(* Logix 5000 project; controller Generic 1768-L43 rev 16.2; software revision 15.01; part 2 of 10 *)
(* tags used below, declared in another part *)
   EL_CTRL_2 : UDT_AxisHistory_CTRL;
   EL_CTRL_3 : UDT_AxisHistory_CTRL;
   EL_CTRL_4 : UDT_AxisHistory_CTRL;
   EventLog_N2 : UDT_AxisHistory_DLM[51];
   EventLog_N3 : UDT_AxisHistory_DLM[51];
   EventLog_N4 : UDT_AxisHistory_DLM[51];
   LogLength : DINT;
   Motion_Group : ALIAS FOR MotionGroup;
   Servo_Axis_Node_2 : ALIAS FOR AXIS_02;
   Servo_Axis_Node_3 : ALIAS FOR AXIS_03;
   Servo_Axis_Node_4 : ALIAS FOR AXIS_04;
(* AXIS_EventLog, continued *)

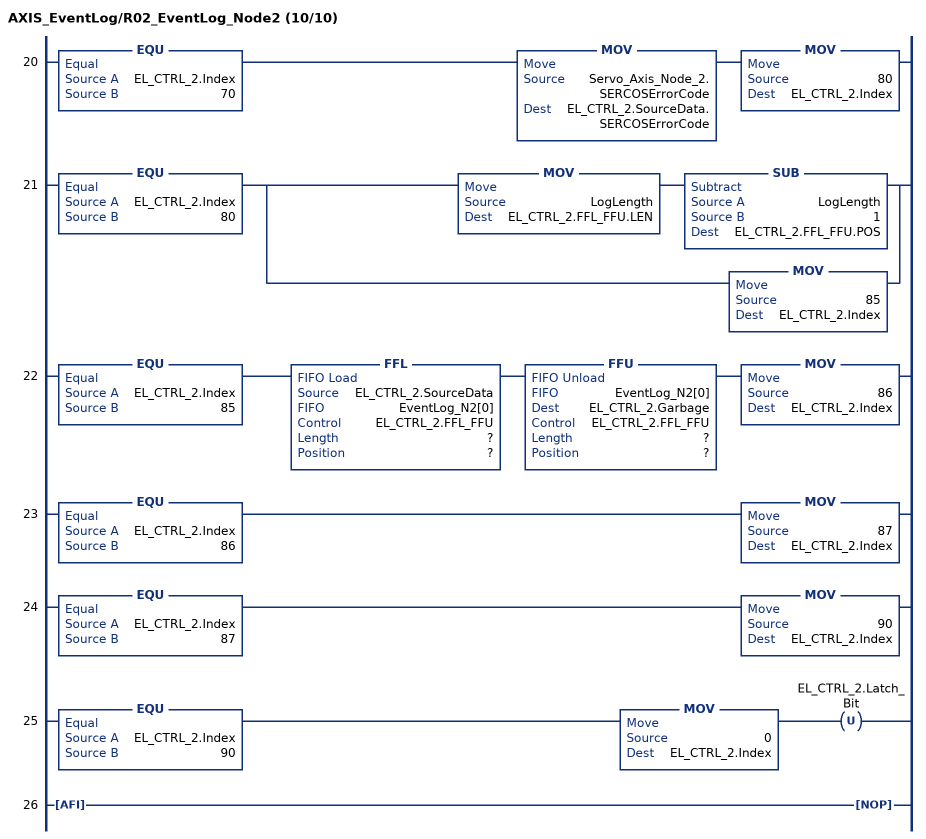
   [picture p36: AXIS_EventLog/R02_EventLog_Node2 rungs 20-26]
   20: EQU(EL_CTRL_2.Index,70)MOV(Servo_Axis_Node_2.SERCOSErrorCode,EL_CTRL_2.SourceData.SERCOSErrorCode)MOV(80,EL_CTRL_2.Index);
   21: EQU(EL_CTRL_2.Index,80)[MOV(LogLength,EL_CTRL_2.FFL_FFU.LEN) SUB(LogLength,1,EL_CTRL_2.FFL_FFU.POS) ,MOV(85,EL_CTRL_2.Index) ];
   22: EQU(EL_CTRL_2.Index,85)FFL(EL_CTRL_2.SourceData,EventLog_N2[0],EL_CTRL_2.FFL_FFU,?,?)FFU(EventLog_N2[0],EL_CTRL_2.Garbage,EL_CTRL_2.FFL_FFU,?,?)MOV(86,EL_CTRL_2.Index);
   23: EQU(EL_CTRL_2.Index,86)MOV(87,EL_CTRL_2.Index);
   24: EQU(EL_CTRL_2.Index,87)MOV(90,EL_CTRL_2.Index);
   25: EQU(EL_CTRL_2.Index,90)MOV(0,EL_CTRL_2.Index)OTU(EL_CTRL_2.Latch_Bit);
   26: AFI()NOP();
END_ROUTINE

ROUTINE R03_EventLog_Node3   (* ladder *)
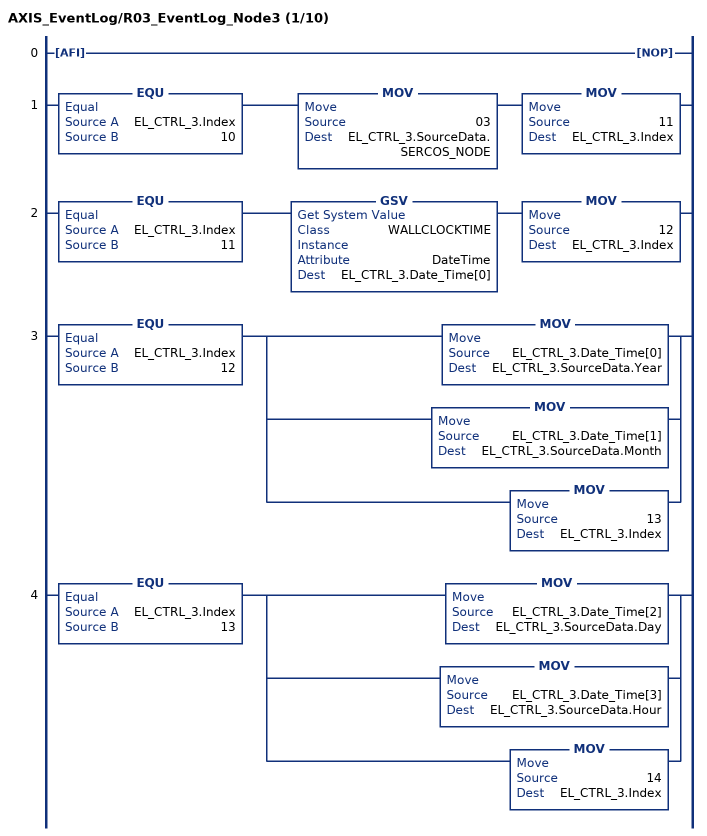
   0: AFI()NOP();
   1: EQU(EL_CTRL_3.Index,10)MOV(03,EL_CTRL_3.SourceData.SERCOS_NODE)MOV(11,EL_CTRL_3.Index);
   2: EQU(EL_CTRL_3.Index,11)GSV(WALLCLOCKTIME,,DateTime,EL_CTRL_3.Date_Time[0])MOV(12,EL_CTRL_3.Index);
   3: EQU(EL_CTRL_3.Index,12)[MOV(EL_CTRL_3.Date_Time[0],EL_CTRL_3.SourceData.Year) ,MOV(EL_CTRL_3.Date_Time[1],EL_CTRL_3.SourceData.Month) ,MOV(13,EL_CTRL_3.Index) ];
   4: EQU(EL_CTRL_3.Index,13)[MOV(EL_CTRL_3.Date_Time[2],EL_CTRL_3.SourceData.Day) ,MOV(EL_CTRL_3.Date_Time[3],EL_CTRL_3.SourceData.Hour) ,MOV(14,EL_CTRL_3.Index) ];
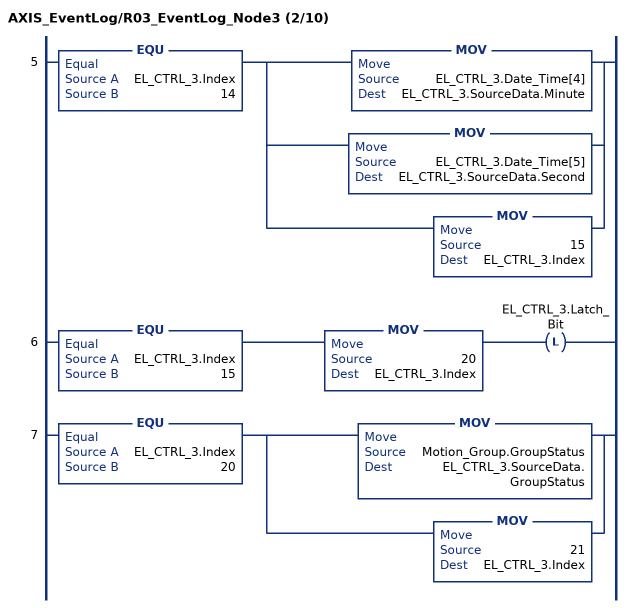
   5: EQU(EL_CTRL_3.Index,14)[MOV(EL_CTRL_3.Date_Time[4],EL_CTRL_3.SourceData.Minute) ,MOV(EL_CTRL_3.Date_Time[5],EL_CTRL_3.SourceData.Second) ,MOV(15,EL_CTRL_3.Index) ];
   6: EQU(EL_CTRL_3.Index,15)MOV(20,EL_CTRL_3.Index)OTL(EL_CTRL_3.Latch_Bit);
   7: EQU(EL_CTRL_3.Index,20)[MOV(Motion_Group.GroupStatus,EL_CTRL_3.SourceData.GroupStatus) ,MOV(21,EL_CTRL_3.Index) ];
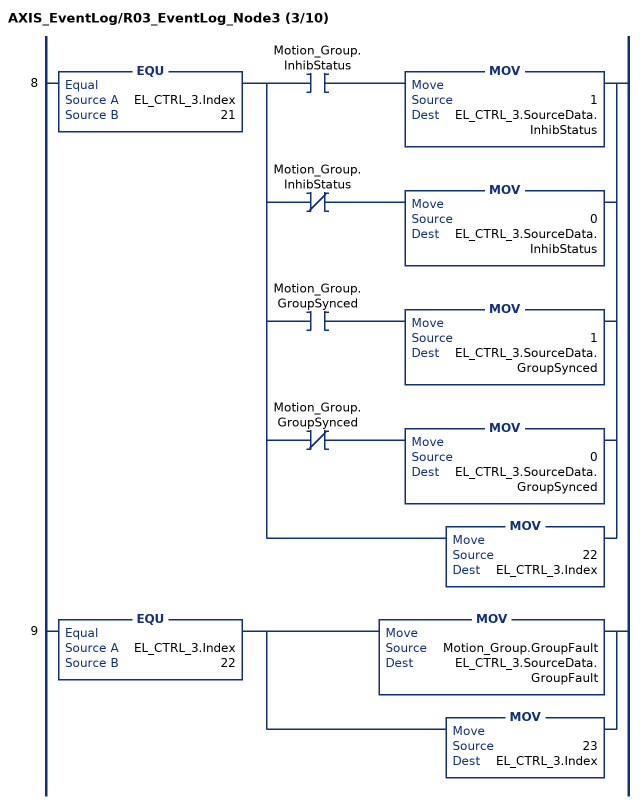
   8: EQU(EL_CTRL_3.Index,21)[XIC(Motion_Group.InhibStatus) MOV(1,EL_CTRL_3.SourceData.InhibStatus) ,XIO(Motion_Group.InhibStatus) MOV(0,EL_CTRL_3.SourceData.InhibStatus) ,XIC(Motion_Group.GroupSynced) MOV(1,EL_CTRL_3.SourceData.GroupSynced) ,XIO(Motion_Group.GroupSynced) MOV(0,EL_CTRL_3.SourceData.GroupSynced) ,MOV(22,EL_CTRL_3.Index) ];
   9: EQU(EL_CTRL_3.Index,22)[MOV(Motion_Group.GroupFault,EL_CTRL_3.SourceData.GroupFault) ,MOV(23,EL_CTRL_3.Index) ];
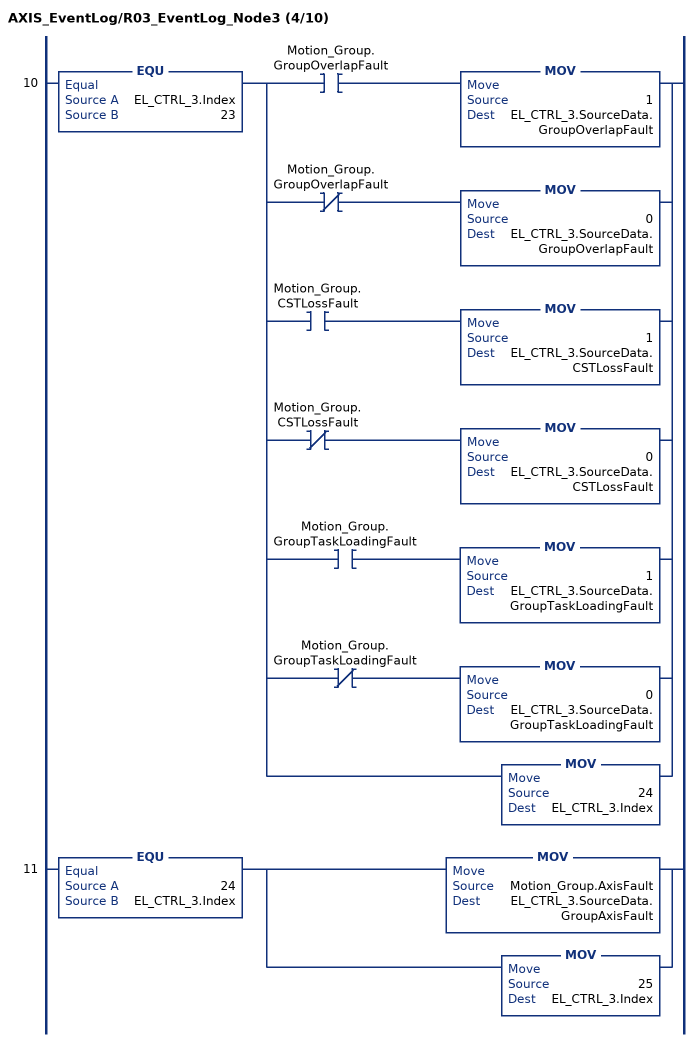
   10: EQU(EL_CTRL_3.Index,23)[XIC(Motion_Group.GroupOverlapFault) MOV(1,EL_CTRL_3.SourceData.GroupOverlapFault) ,XIO(Motion_Group.GroupOverlapFault) MOV(0,EL_CTRL_3.SourceData.GroupOverlapFault) ,XIC(Motion_Group.CSTLossFault) MOV(1,EL_CTRL_3.SourceData.CSTLossFault) ,XIO(Motion_Group.CSTLossFault) MOV(0,EL_CTRL_3.SourceData.CSTLossFault) ,XIC(Motion_Group.GroupTaskLoadingFault) MOV(1,EL_CTRL_3.SourceData.GroupTaskLoadingFault) ,XIO(Motion_Group.GroupTaskLoadingFault) MOV(0,EL_CTRL_3.SourceData.GroupTaskLoadingFault) ,MOV(24,EL_CTRL_3.Index) ];
   11: EQU(24,EL_CTRL_3.Index)[MOV(Motion_Group.AxisFault,EL_CTRL_3.SourceData.GroupAxisFault) ,MOV(25,EL_CTRL_3.Index) ];
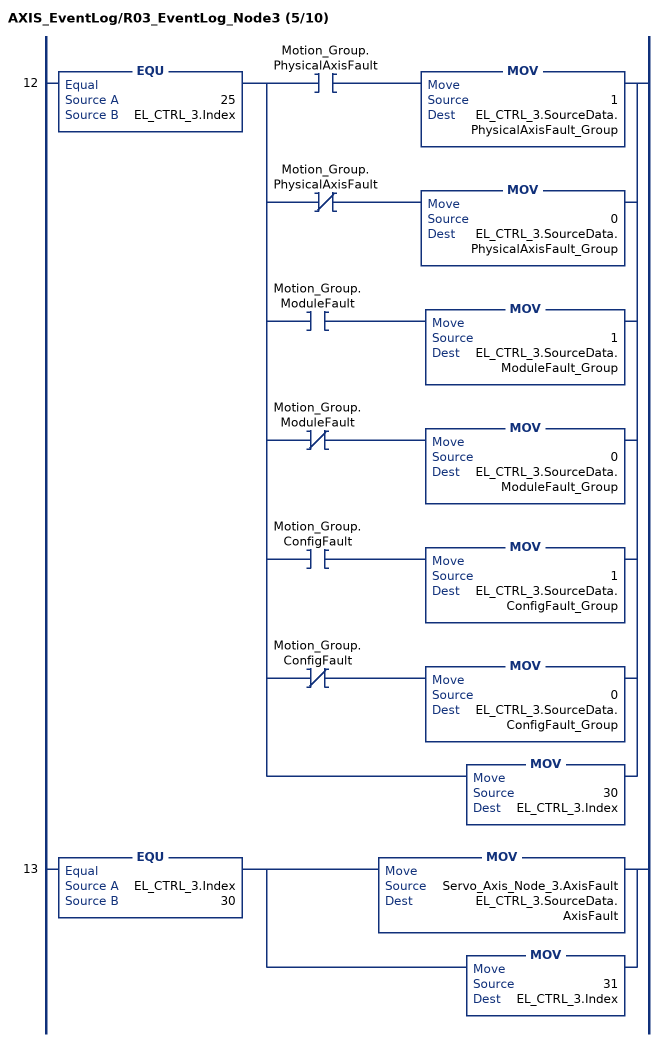
   12: EQU(25,EL_CTRL_3.Index)[XIC(Motion_Group.PhysicalAxisFault) MOV(1,EL_CTRL_3.SourceData.PhysicalAxisFault_Group) ,XIO(Motion_Group.PhysicalAxisFault) MOV(0,EL_CTRL_3.SourceData.PhysicalAxisFault_Group) ,XIC(Motion_Group.ModuleFault) MOV(1,EL_CTRL_3.SourceData.ModuleFault_Group) ,XIO(Motion_Group.ModuleFault) MOV(0,EL_CTRL_3.SourceData.ModuleFault_Group) ,XIC(Motion_Group.ConfigFault) MOV(1,EL_CTRL_3.SourceData.ConfigFault_Group) ,XIO(Motion_Group.ConfigFault) MOV(0,EL_CTRL_3.SourceData.ConfigFault_Group) ,MOV(30,EL_CTRL_3.Index) ];
   13: EQU(EL_CTRL_3.Index,30)[MOV(Servo_Axis_Node_3.AxisFault,EL_CTRL_3.SourceData.AxisFault) ,MOV(31,EL_CTRL_3.Index) ];
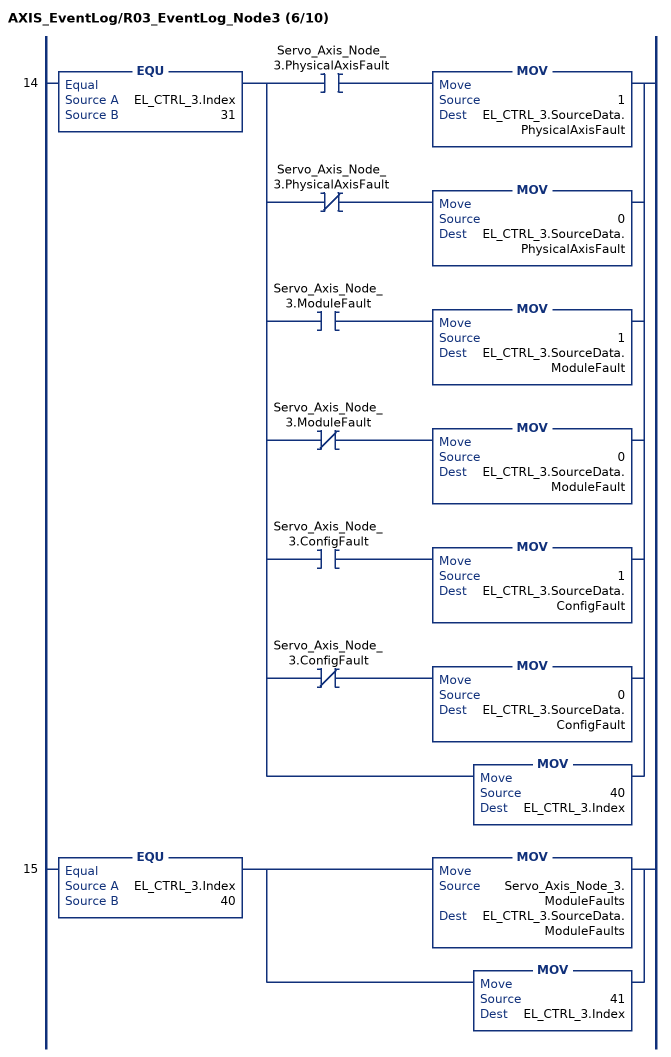
   14: EQU(EL_CTRL_3.Index,31)[XIC(Servo_Axis_Node_3.PhysicalAxisFault) MOV(1,EL_CTRL_3.SourceData.PhysicalAxisFault) ,XIO(Servo_Axis_Node_3.PhysicalAxisFault) MOV(0,EL_CTRL_3.SourceData.PhysicalAxisFault) ,XIC(Servo_Axis_Node_3.ModuleFault) MOV(1,EL_CTRL_3.SourceData.ModuleFault) ,XIO(Servo_Axis_Node_3.ModuleFault) MOV(0,EL_CTRL_3.SourceData.ModuleFault) ,XIC(Servo_Axis_Node_3.ConfigFault) MOV(1,EL_CTRL_3.SourceData.ConfigFault) ,XIO(Servo_Axis_Node_3.ConfigFault) MOV(0,EL_CTRL_3.SourceData.ConfigFault) ,MOV(40,EL_CTRL_3.Index) ];
   15: EQU(EL_CTRL_3.Index,40)[MOV(Servo_Axis_Node_3.ModuleFaults,EL_CTRL_3.SourceData.ModuleFaults) ,MOV(41,EL_CTRL_3.Index) ];
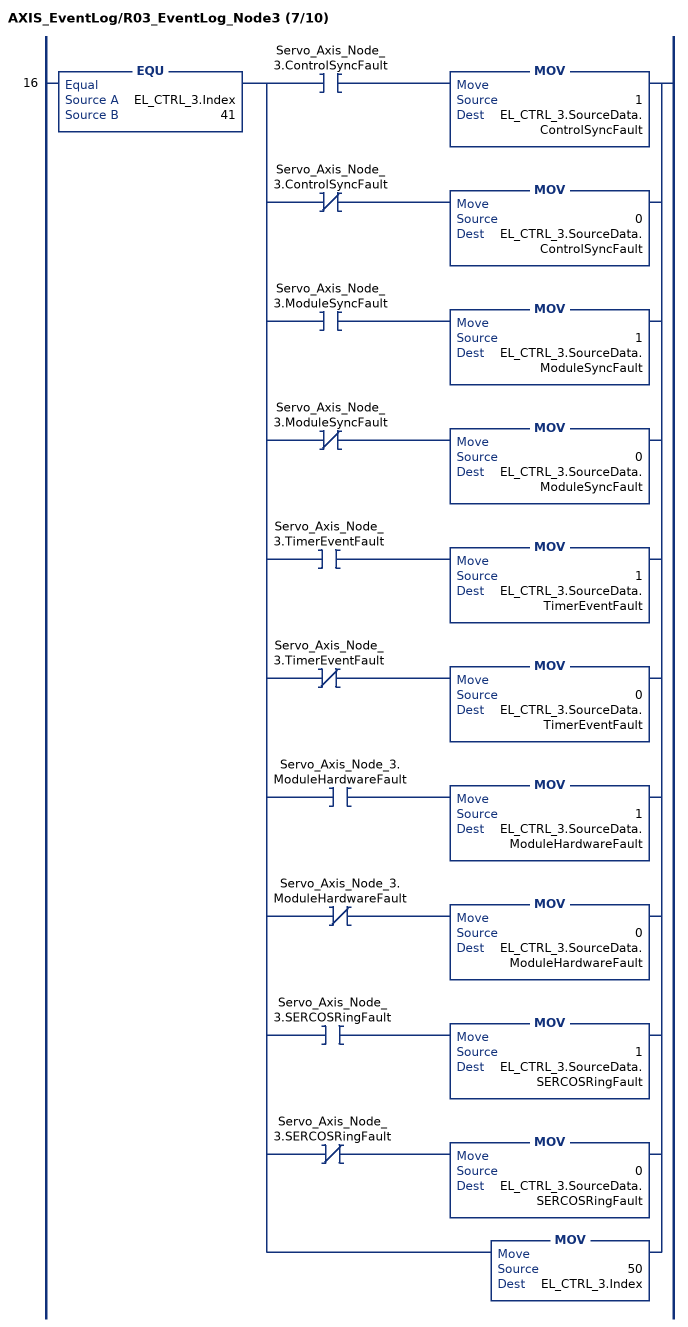
   16: EQU(EL_CTRL_3.Index,41)[XIC(Servo_Axis_Node_3.ControlSyncFault) MOV(1,EL_CTRL_3.SourceData.ControlSyncFault) ,XIO(Servo_Axis_Node_3.ControlSyncFault) MOV(0,EL_CTRL_3.SourceData.ControlSyncFault) ,XIC(Servo_Axis_Node_3.ModuleSyncFault) MOV(1,EL_CTRL_3.SourceData.ModuleSyncFault) ,XIO(Servo_Axis_Node_3.ModuleSyncFault) MOV(0,EL_CTRL_3.SourceData.ModuleSyncFault) ,XIC(Servo_Axis_Node_3.TimerEventFault) MOV(1,EL_CTRL_3.SourceData.TimerEventFault) ,XIO(Servo_Axis_Node_3.TimerEventFault) MOV(0,EL_CTRL_3.SourceData.TimerEventFault) ,XIC(Servo_Axis_Node_3.ModuleHardwareFault) MOV(1,EL_CTRL_3.SourceData.ModuleHardwareFault) ,XIO(Servo_Axis_Node_3.ModuleHardwareFault) MOV(0,EL_CTRL_3.SourceData.ModuleHardwareFault) ,XIC(Servo_Axis_Node_3.SERCOSRingFault) MOV(1,EL_CTRL_3.SourceData.SERCOSRingFault) ,XIO(Servo_Axis_Node_3.SERCOSRingFault) MOV(0,EL_CTRL_3.SourceData.SERCOSRingFault) ,MOV(50,EL_CTRL_3.Index) ];
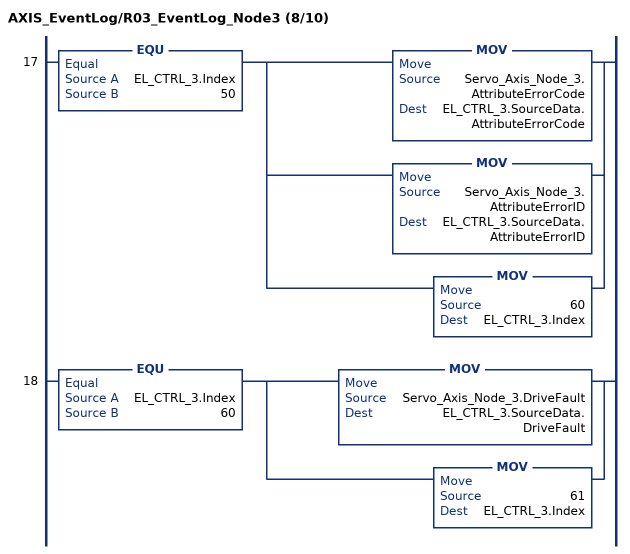
   17: EQU(EL_CTRL_3.Index,50)[MOV(Servo_Axis_Node_3.AttributeErrorCode,EL_CTRL_3.SourceData.AttributeErrorCode) ,MOV(Servo_Axis_Node_3.AttributeErrorID,EL_CTRL_3.SourceData.AttributeErrorID) ,MOV(60,EL_CTRL_3.Index) ];
   18: EQU(EL_CTRL_3.Index,60)[MOV(Servo_Axis_Node_3.DriveFault,EL_CTRL_3.SourceData.DriveFault) ,MOV(61,EL_CTRL_3.Index) ];
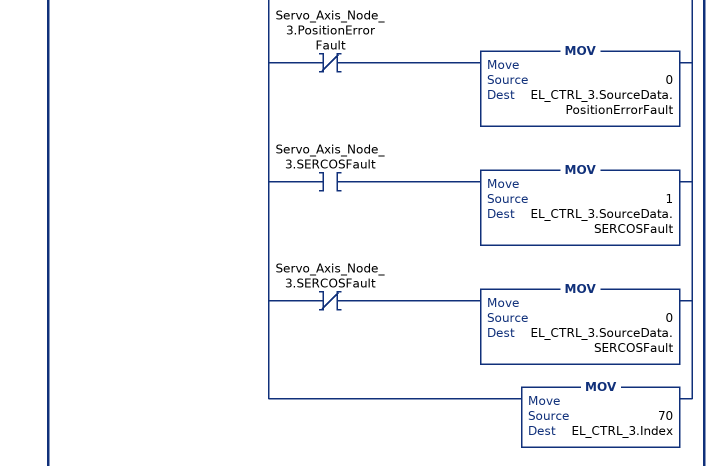
   19: EQU(EL_CTRL_3.Index,61)[XIC(Servo_Axis_Node_3.PosSoftOvertravelFault) MOV(1,EL_CTRL_3.SourceData.PosSoftOvertravelFault) ,XIO(Servo_Axis_Node_3.PosSoftOvertravelFault) MOV(0,EL_CTRL_3.SourceData.PosSoftOvertravelFault) ,XIC(Servo_Axis_Node_3.NegSoftOvertravelFault) MOV(1,EL_CTRL_3.SourceData.NegSoftOvertravelFault) ,XIO(Servo_Axis_Node_3.NegSoftOvertravelFault) MOV(0,EL_CTRL_3.SourceData.NegSoftOvertravelFault) ,XIC(Servo_Axis_Node_3.PosHardOvertravelFault) MOV(1,EL_CTRL_3.SourceData.PosHardOvertravelFault) ,XIO(Servo_Axis_Node_3.PosHardOvertravelFault) MOV(0,EL_CTRL_3.SourceData.PosHardOvertravelFault) ,XIC(Servo_Axis_Node_3.NegHardOvertravelFault) MOV(1,EL_CTRL_3.SourceData.NegHardOvertravelFault) ,XIO(Servo_Axis_Node_3.NegHardOvertravelFault) MOV(0,EL_CTRL_3.SourceData.NegHardOvertravelFault) ,XIC(Servo_Axis_Node_3.MotFeedbackFault) MOV(1,EL_CTRL_3.SourceData.MotFeedbackFault) ,XIO(Servo_Axis_Node_3.MotFeedbackFault) MOV(0,EL_CTRL_3.SourceData.MotFeedbackFault) ,XIC(Servo_Axis_Node_3.MotFeedbackNoiseFault) MOV(1,EL_CTRL_3.SourceData.MotFeedbackNoiseFault) ,XIO(Servo_Axis_Node_3.MotFeedbackNoiseFault) MOV(0,EL_CTRL_3.SourceData.MotFeedbackNoiseFault) ,XIC(Servo_Axis_Node_3.AuxFeedbackFault) MOV(1,EL_CTRL_3.SourceData.AuxFeedbackFault) ,XIO(Servo_Axis_Node_3.AuxFeedbackFault) MOV(0,EL_CTRL_3.SourceData.AuxFeedbackFault) ,XIC(Servo_Axis_Node_3.AuxFeedbackNoiseFault) MOV(1,EL_CTRL_3.SourceData.AuxFeedbackNoiseFault) ,XIO(Servo_Axis_Node_3.AuxFeedbackNoiseFault) MOV(0,EL_CTRL_3.SourceData.AuxFeedbackNoiseFault) ,XIC(Servo_Axis_Node_3.DriveEnableInputFault) MOV(1,EL_CTRL_3.SourceData.DriveEnableInputFault) ,XIO(Servo_Axis_Node_3.DriveEnableInputFault) MOV(0,EL_CTRL_3.SourceData.DriveEnableInputFault) ,XIC(Servo_Axis_Node_3.CommonBusFault) MOV(1,EL_CTRL_3.SourceData.CommonBusFault) ,XIO(Servo_Axis_Node_3.CommonBusFault) MOV(0,EL_CTRL_3.SourceData.CommonBusFault) ,XIC(Servo_Axis_Node_3.PreChargeOverloadFault) MOV(1,EL_CTRL_3.SourceData.PreChargeOverloadFault) ,XIO(Servo_Axis_Node_3.PreChargeOverloadFault) MOV(0,EL_CTRL_3.SourceData.PreChargeOverloadFault) ,XIC(Servo_Axis_Node_3.GroundShortFault) MOV(1,EL_CTRL_3.SourceData.GroundShortFault) ,XIO(Servo_Axis_Node_3.GroundShortFault) MOV(0,EL_CTRL_3.SourceData.GroundShortFault) ,XIC(Servo_Axis_Node_3.DriveHardFault) MOV(1,EL_CTRL_3.SourceData.DriveHardFault) ,XIO(Servo_Axis_Node_3.DriveHardFault) MOV(0,EL_CTRL_3.SourceData.DriveHardFault) ,XIC(Servo_Axis_Node_3.OverSpeedFault) MOV(1,EL_CTRL_3.SourceData.OverSpeedFault) ,XIO(Servo_Axis_Node_3.OverSpeedFault) MOV(0,EL_CTRL_3.SourceData.OverSpeedFault) ,XIC(Servo_Axis_Node_3.OverloadFault) MOV(1,EL_CTRL_3.SourceData.OverloadFault) ,XIO(Servo_Axis_Node_3.OverloadFault) MOV(0,EL_CTRL_3.SourceData.OverloadFault) ,XIC(Servo_Axis_Node_3.DriveOvertempFault) MOV(1,EL_CTRL_3.SourceData.DriveOvertempFault) ,XIO(Servo_Axis_Node_3.DriveOvertempFault) MOV(0,EL_CTRL_3.SourceData.DriveOvertempFault) ,XIC(Servo_Axis_Node_3.MotorOvertempFault) MOV(1,EL_CTRL_3.SourceData.MotorOvertempFault) ,XIO(Servo_Axis_Node_3.MotorOvertempFault) MOV(0,EL_CTRL_3.SourceData.MotorOvertempFault) ,XIC(Servo_Axis_Node_3.DriveCoolingFault) MOV(1,EL_CTRL_3.SourceData.DriveCoolingFault) ,XIO(Servo_Axis_Node_3.DriveCoolingFault) MOV(0,EL_CTRL_3.SourceData.DriveCoolingFault) ,XIC(Servo_Axis_Node_3.DriveControlVoltageFault) MOV(1,EL_CTRL_3.SourceData.DriveControlVoltageFault) ,XIO(Servo_Axis_Node_3.DriveControlVoltageFault) MOV(0,EL_CTRL_3.SourceData.DriveControlVoltageFault) ,XIC(Servo_Axis_Node_3.FeedbackFault) MOV(1,EL_CTRL_3.SourceData.FeedbackFault) ,XIO(Servo_Axis_Node_3.FeedbackFault) MOV(0,EL_CTRL_3.SourceData.FeedbackFault) ,XIC(Servo_Axis_Node_3.CommutationFault) MOV(1,EL_CTRL_3.SourceData.CommutationFault) ,XIO(Servo_Axis_Node_3.CommutationFault) MOV(0,EL_CTRL_3.SourceData.CommutationFault) ,XIC(Servo_Axis_Node_3.DriveOvercurrentFault) MOV(1,EL_CTRL_3.SourceData.DriveOvercurrentFault) ,XIO(Servo_Axis_Node_3.DriveOvercurrentFault) MOV(0,EL_CTRL_3.SourceData.DriveOvercurrentFault) ,XIC(Servo_Axis_Node_3.DriveOvervoltageFault) MOV(1,EL_CTRL_3.SourceData.DriveOvervoltageFault) ,XIO(Servo_Axis_Node_3.DriveOvervoltageFault) MOV(0,EL_CTRL_3.SourceData.DriveOvervoltageFault) ,XIC(Servo_Axis_Node_3.DriveUndervoltageFault) MOV(1,EL_CTRL_3.SourceData.DriveUndervoltageFault) ,XIO(Servo_Axis_Node_3.DriveUndervoltageFault) MOV(0,EL_CTRL_3.SourceData.DriveUndervoltageFault) ,XIC(Servo_Axis_Node_3.PowerPhaseLossFault) MOV(1,EL_CTRL_3.SourceData.PowerPhaseLossFault) ,XIO(Servo_Axis_Node_3.PowerPhaseLossFault) MOV(0,EL_CTRL_3.SourceData.PowerPhaseLossFault) ,XIC(Servo_Axis_Node_3.PositionErrorFault) MOV(1,EL_CTRL_3.SourceData.PositionErrorFault) ,XIO(Servo_Axis_Node_3.PositionErrorFault) MOV(0,EL_CTRL_3.SourceData.PositionErrorFault) ,XIC(Servo_Axis_Node_3.SERCOSFault) MOV(1,EL_CTRL_3.SourceData.SERCOSFault) ,XIO(Servo_Axis_Node_3.SERCOSFault) MOV(0,EL_CTRL_3.SourceData.SERCOSFault) ,MOV(70,EL_CTRL_3.Index) ];
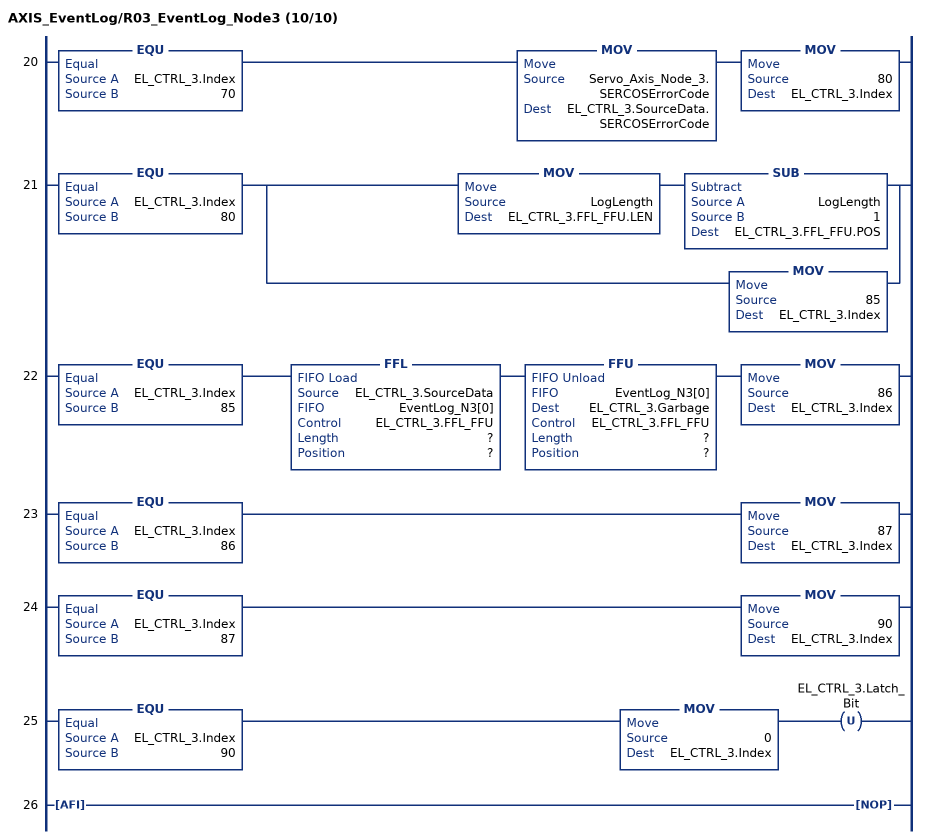
   20: EQU(EL_CTRL_3.Index,70)MOV(Servo_Axis_Node_3.SERCOSErrorCode,EL_CTRL_3.SourceData.SERCOSErrorCode)MOV(80,EL_CTRL_3.Index);
   21: EQU(EL_CTRL_3.Index,80)[MOV(LogLength,EL_CTRL_3.FFL_FFU.LEN) SUB(LogLength,1,EL_CTRL_3.FFL_FFU.POS) ,MOV(85,EL_CTRL_3.Index) ];
   22: EQU(EL_CTRL_3.Index,85)FFL(EL_CTRL_3.SourceData,EventLog_N3[0],EL_CTRL_3.FFL_FFU,?,?)FFU(EventLog_N3[0],EL_CTRL_3.Garbage,EL_CTRL_3.FFL_FFU,?,?)MOV(86,EL_CTRL_3.Index);
   23: EQU(EL_CTRL_3.Index,86)MOV(87,EL_CTRL_3.Index);
   24: EQU(EL_CTRL_3.Index,87)MOV(90,EL_CTRL_3.Index);
   25: EQU(EL_CTRL_3.Index,90)MOV(0,EL_CTRL_3.Index)OTU(EL_CTRL_3.Latch_Bit);
   26: AFI()NOP();
END_ROUTINE

ROUTINE R04_EventLog_Node4   (* ladder *)
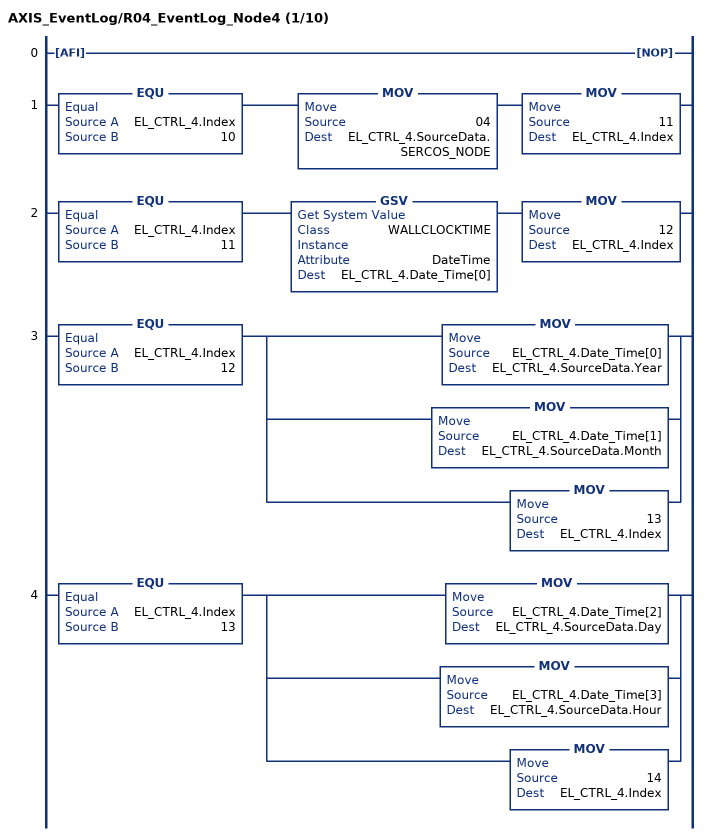
   0: AFI()NOP();
   1: EQU(EL_CTRL_4.Index,10)MOV(04,EL_CTRL_4.SourceData.SERCOS_NODE)MOV(11,EL_CTRL_4.Index);
   2: EQU(EL_CTRL_4.Index,11)GSV(WALLCLOCKTIME,,DateTime,EL_CTRL_4.Date_Time[0])MOV(12,EL_CTRL_4.Index);
   3: EQU(EL_CTRL_4.Index,12)[MOV(EL_CTRL_4.Date_Time[0],EL_CTRL_4.SourceData.Year) ,MOV(EL_CTRL_4.Date_Time[1],EL_CTRL_4.SourceData.Month) ,MOV(13,EL_CTRL_4.Index) ];
   4: EQU(EL_CTRL_4.Index,13)[MOV(EL_CTRL_4.Date_Time[2],EL_CTRL_4.SourceData.Day) ,MOV(EL_CTRL_4.Date_Time[3],EL_CTRL_4.SourceData.Hour) ,MOV(14,EL_CTRL_4.Index) ];
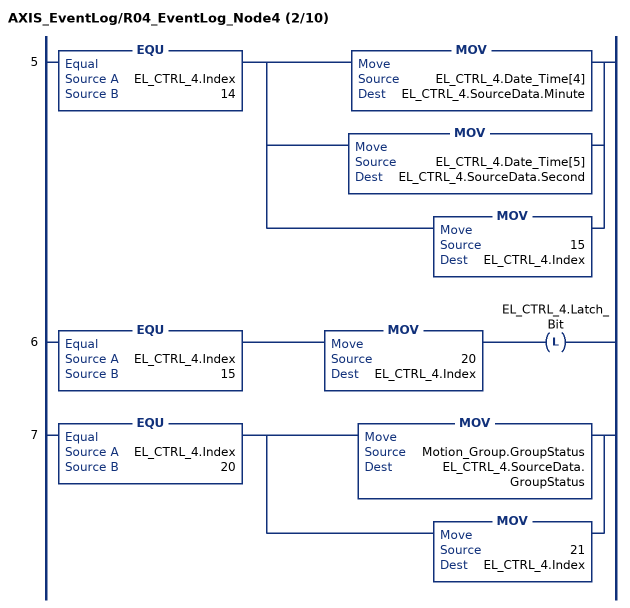
   5: EQU(EL_CTRL_4.Index,14)[MOV(EL_CTRL_4.Date_Time[4],EL_CTRL_4.SourceData.Minute) ,MOV(EL_CTRL_4.Date_Time[5],EL_CTRL_4.SourceData.Second) ,MOV(15,EL_CTRL_4.Index) ];
   6: EQU(EL_CTRL_4.Index,15)MOV(20,EL_CTRL_4.Index)OTL(EL_CTRL_4.Latch_Bit);
   7: EQU(EL_CTRL_4.Index,20)[MOV(Motion_Group.GroupStatus,EL_CTRL_4.SourceData.GroupStatus) ,MOV(21,EL_CTRL_4.Index) ];
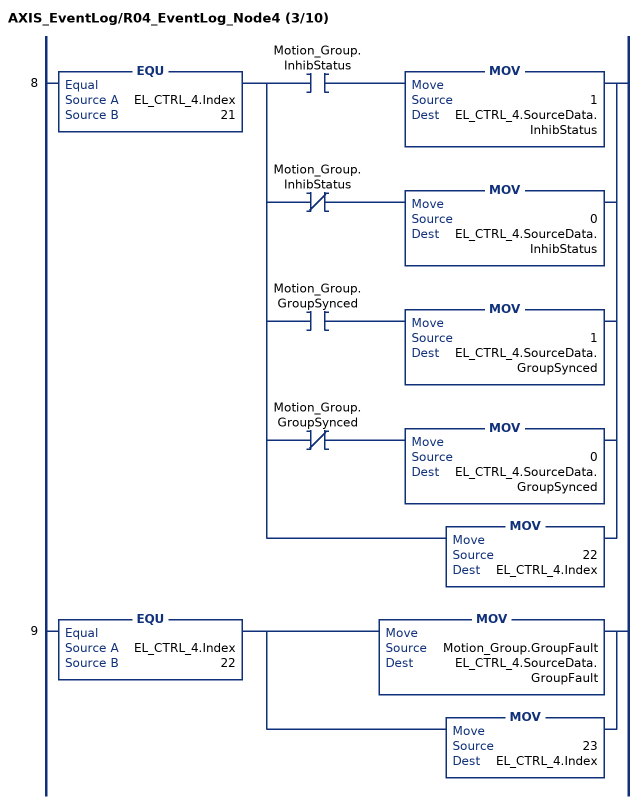
   8: EQU(EL_CTRL_4.Index,21)[XIC(Motion_Group.InhibStatus) MOV(1,EL_CTRL_4.SourceData.InhibStatus) ,XIO(Motion_Group.InhibStatus) MOV(0,EL_CTRL_4.SourceData.InhibStatus) ,XIC(Motion_Group.GroupSynced) MOV(1,EL_CTRL_4.SourceData.GroupSynced) ,XIO(Motion_Group.GroupSynced) MOV(0,EL_CTRL_4.SourceData.GroupSynced) ,MOV(22,EL_CTRL_4.Index) ];
   9: EQU(EL_CTRL_4.Index,22)[MOV(Motion_Group.GroupFault,EL_CTRL_4.SourceData.GroupFault) ,MOV(23,EL_CTRL_4.Index) ];
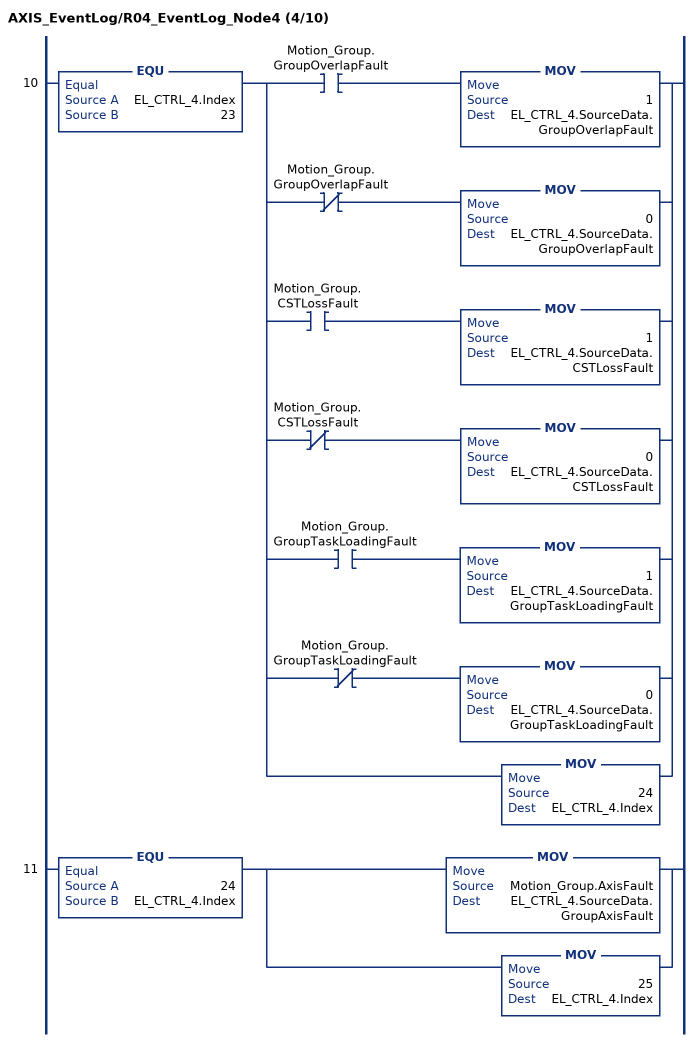
   10: EQU(EL_CTRL_4.Index,23)[XIC(Motion_Group.GroupOverlapFault) MOV(1,EL_CTRL_4.SourceData.GroupOverlapFault) ,XIO(Motion_Group.GroupOverlapFault) MOV(0,EL_CTRL_4.SourceData.GroupOverlapFault) ,XIC(Motion_Group.CSTLossFault) MOV(1,EL_CTRL_4.SourceData.CSTLossFault) ,XIO(Motion_Group.CSTLossFault) MOV(0,EL_CTRL_4.SourceData.CSTLossFault) ,XIC(Motion_Group.GroupTaskLoadingFault) MOV(1,EL_CTRL_4.SourceData.GroupTaskLoadingFault) ,XIO(Motion_Group.GroupTaskLoadingFault) MOV(0,EL_CTRL_4.SourceData.GroupTaskLoadingFault) ,MOV(24,EL_CTRL_4.Index) ];
   11: EQU(24,EL_CTRL_4.Index)[MOV(Motion_Group.AxisFault,EL_CTRL_4.SourceData.GroupAxisFault) ,MOV(25,EL_CTRL_4.Index) ];
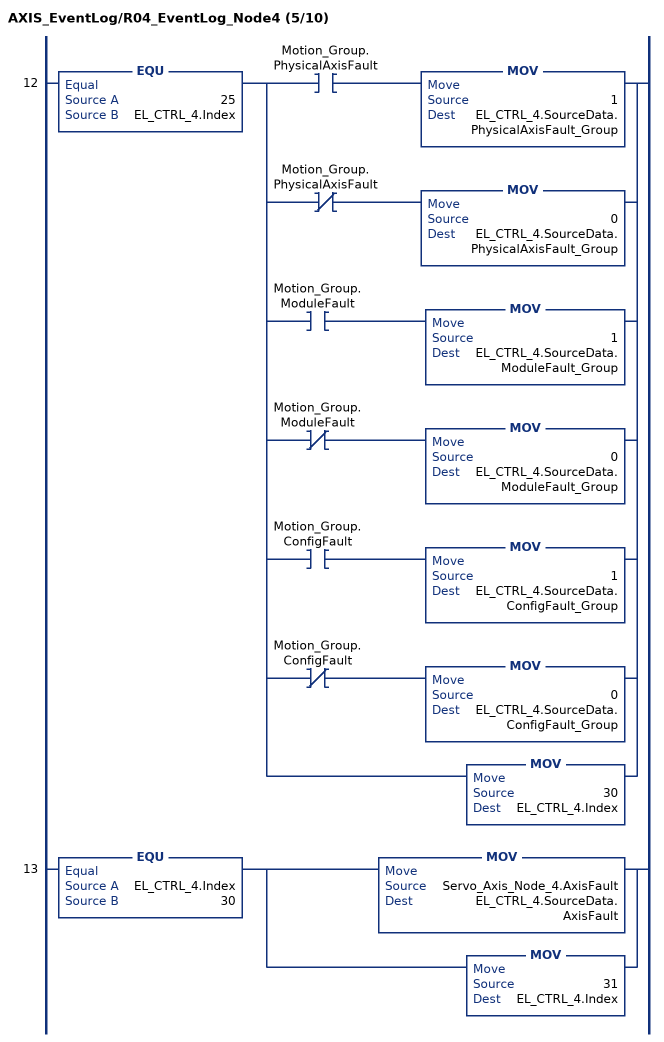
   12: EQU(25,EL_CTRL_4.Index)[XIC(Motion_Group.PhysicalAxisFault) MOV(1,EL_CTRL_4.SourceData.PhysicalAxisFault_Group) ,XIO(Motion_Group.PhysicalAxisFault) MOV(0,EL_CTRL_4.SourceData.PhysicalAxisFault_Group) ,XIC(Motion_Group.ModuleFault) MOV(1,EL_CTRL_4.SourceData.ModuleFault_Group) ,XIO(Motion_Group.ModuleFault) MOV(0,EL_CTRL_4.SourceData.ModuleFault_Group) ,XIC(Motion_Group.ConfigFault) MOV(1,EL_CTRL_4.SourceData.ConfigFault_Group) ,XIO(Motion_Group.ConfigFault) MOV(0,EL_CTRL_4.SourceData.ConfigFault_Group) ,MOV(30,EL_CTRL_4.Index) ];
   13: EQU(EL_CTRL_4.Index,30)[MOV(Servo_Axis_Node_4.AxisFault,EL_CTRL_4.SourceData.AxisFault) ,MOV(31,EL_CTRL_4.Index) ];
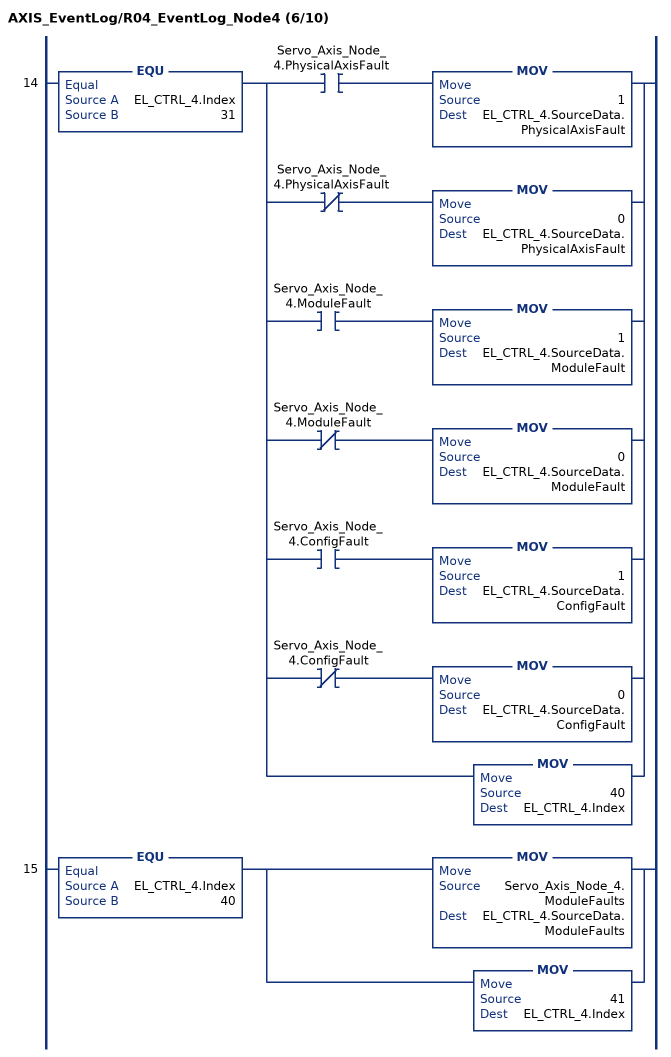
   14: EQU(EL_CTRL_4.Index,31)[XIC(Servo_Axis_Node_4.PhysicalAxisFault) MOV(1,EL_CTRL_4.SourceData.PhysicalAxisFault) ,XIO(Servo_Axis_Node_4.PhysicalAxisFault) MOV(0,EL_CTRL_4.SourceData.PhysicalAxisFault) ,XIC(Servo_Axis_Node_4.ModuleFault) MOV(1,EL_CTRL_4.SourceData.ModuleFault) ,XIO(Servo_Axis_Node_4.ModuleFault) MOV(0,EL_CTRL_4.SourceData.ModuleFault) ,XIC(Servo_Axis_Node_4.ConfigFault) MOV(1,EL_CTRL_4.SourceData.ConfigFault) ,XIO(Servo_Axis_Node_4.ConfigFault) MOV(0,EL_CTRL_4.SourceData.ConfigFault) ,MOV(40,EL_CTRL_4.Index) ];
   15: EQU(EL_CTRL_4.Index,40)[MOV(Servo_Axis_Node_4.ModuleFaults,EL_CTRL_4.SourceData.ModuleFaults) ,MOV(41,EL_CTRL_4.Index) ];
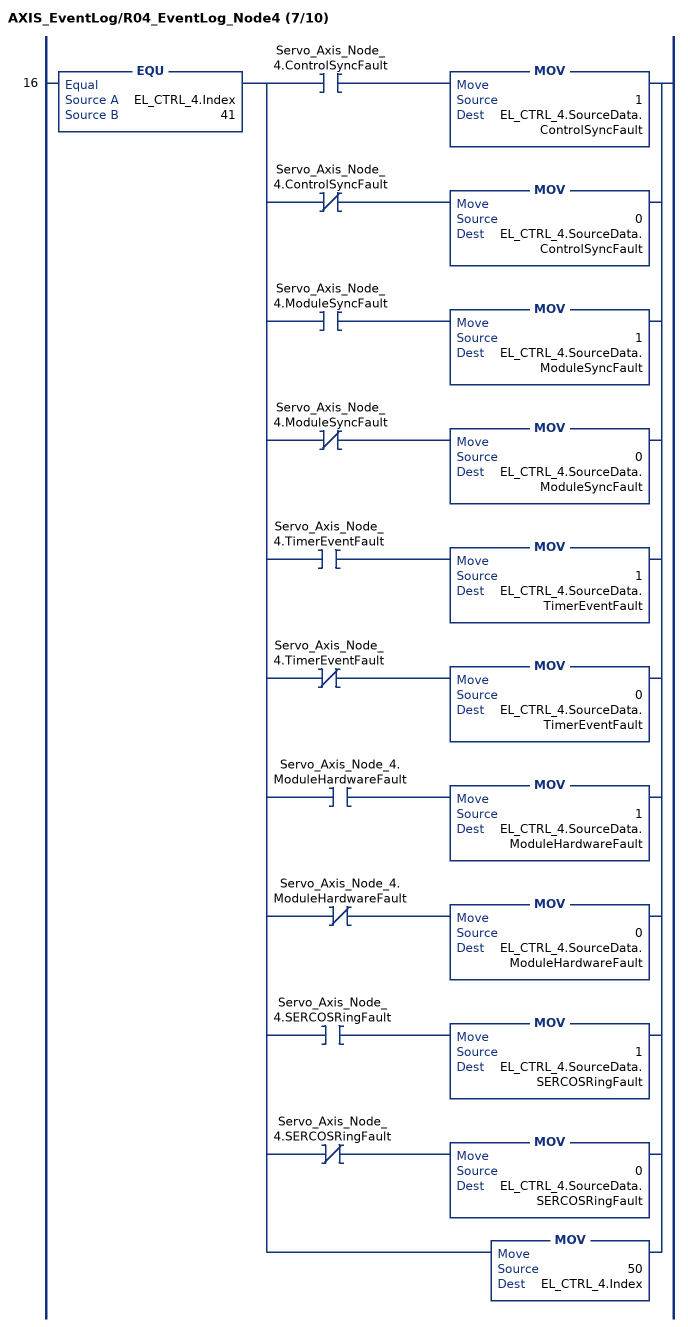
   16: EQU(EL_CTRL_4.Index,41)[XIC(Servo_Axis_Node_4.ControlSyncFault) MOV(1,EL_CTRL_4.SourceData.ControlSyncFault) ,XIO(Servo_Axis_Node_4.ControlSyncFault) MOV(0,EL_CTRL_4.SourceData.ControlSyncFault) ,XIC(Servo_Axis_Node_4.ModuleSyncFault) MOV(1,EL_CTRL_4.SourceData.ModuleSyncFault) ,XIO(Servo_Axis_Node_4.ModuleSyncFault) MOV(0,EL_CTRL_4.SourceData.ModuleSyncFault) ,XIC(Servo_Axis_Node_4.TimerEventFault) MOV(1,EL_CTRL_4.SourceData.TimerEventFault) ,XIO(Servo_Axis_Node_4.TimerEventFault) MOV(0,EL_CTRL_4.SourceData.TimerEventFault) ,XIC(Servo_Axis_Node_4.ModuleHardwareFault) MOV(1,EL_CTRL_4.SourceData.ModuleHardwareFault) ,XIO(Servo_Axis_Node_4.ModuleHardwareFault) MOV(0,EL_CTRL_4.SourceData.ModuleHardwareFault) ,XIC(Servo_Axis_Node_4.SERCOSRingFault) MOV(1,EL_CTRL_4.SourceData.SERCOSRingFault) ,XIO(Servo_Axis_Node_4.SERCOSRingFault) MOV(0,EL_CTRL_4.SourceData.SERCOSRingFault) ,MOV(50,EL_CTRL_4.Index) ];
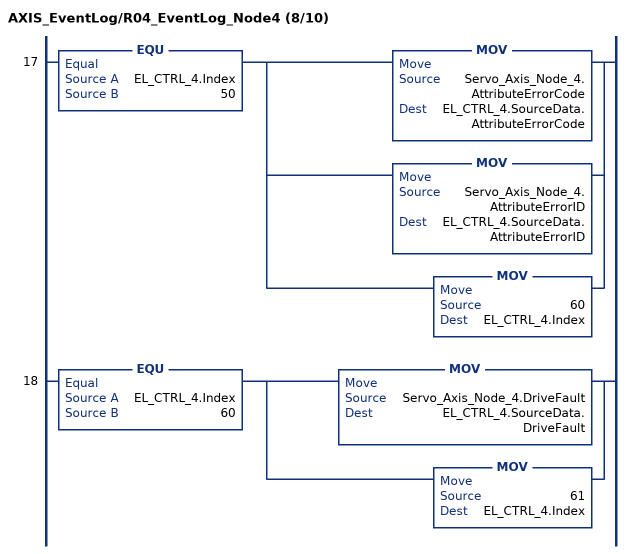
   17: EQU(EL_CTRL_4.Index,50)[MOV(Servo_Axis_Node_4.AttributeErrorCode,EL_CTRL_4.SourceData.AttributeErrorCode) ,MOV(Servo_Axis_Node_4.AttributeErrorID,EL_CTRL_4.SourceData.AttributeErrorID) ,MOV(60,EL_CTRL_4.Index) ];
   18: EQU(EL_CTRL_4.Index,60)[MOV(Servo_Axis_Node_4.DriveFault,EL_CTRL_4.SourceData.DriveFault) ,MOV(61,EL_CTRL_4.Index) ];
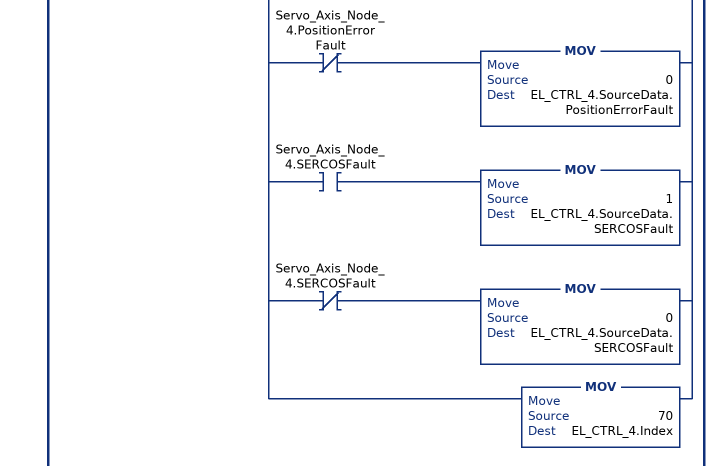
   19: EQU(EL_CTRL_4.Index,61)[XIC(Servo_Axis_Node_4.PosSoftOvertravelFault) MOV(1,EL_CTRL_4.SourceData.PosSoftOvertravelFault) ,XIO(Servo_Axis_Node_4.PosSoftOvertravelFault) MOV(0,EL_CTRL_4.SourceData.PosSoftOvertravelFault) ,XIC(Servo_Axis_Node_4.NegSoftOvertravelFault) MOV(1,EL_CTRL_4.SourceData.NegSoftOvertravelFault) ,XIO(Servo_Axis_Node_4.NegSoftOvertravelFault) MOV(0,EL_CTRL_4.SourceData.NegSoftOvertravelFault) ,XIC(Servo_Axis_Node_4.PosHardOvertravelFault) MOV(1,EL_CTRL_4.SourceData.PosHardOvertravelFault) ,XIO(Servo_Axis_Node_4.PosHardOvertravelFault) MOV(0,EL_CTRL_4.SourceData.PosHardOvertravelFault) ,XIC(Servo_Axis_Node_4.NegHardOvertravelFault) MOV(1,EL_CTRL_4.SourceData.NegHardOvertravelFault) ,XIO(Servo_Axis_Node_4.NegHardOvertravelFault) MOV(0,EL_CTRL_4.SourceData.NegHardOvertravelFault) ,XIC(Servo_Axis_Node_4.MotFeedbackFault) MOV(1,EL_CTRL_4.SourceData.MotFeedbackFault) ,XIO(Servo_Axis_Node_4.MotFeedbackFault) MOV(0,EL_CTRL_4.SourceData.MotFeedbackFault) ,XIC(Servo_Axis_Node_4.MotFeedbackNoiseFault) MOV(1,EL_CTRL_4.SourceData.MotFeedbackNoiseFault) ,XIO(Servo_Axis_Node_4.MotFeedbackNoiseFault) MOV(0,EL_CTRL_4.SourceData.MotFeedbackNoiseFault) ,XIC(Servo_Axis_Node_4.AuxFeedbackFault) MOV(1,EL_CTRL_4.SourceData.AuxFeedbackFault) ,XIO(Servo_Axis_Node_4.AuxFeedbackFault) MOV(0,EL_CTRL_4.SourceData.AuxFeedbackFault) ,XIC(Servo_Axis_Node_4.AuxFeedbackNoiseFault) MOV(1,EL_CTRL_4.SourceData.AuxFeedbackNoiseFault) ,XIO(Servo_Axis_Node_4.AuxFeedbackNoiseFault) MOV(0,EL_CTRL_4.SourceData.AuxFeedbackNoiseFault) ,XIC(Servo_Axis_Node_4.DriveEnableInputFault) MOV(1,EL_CTRL_4.SourceData.DriveEnableInputFault) ,XIO(Servo_Axis_Node_4.DriveEnableInputFault) MOV(0,EL_CTRL_4.SourceData.DriveEnableInputFault) ,XIC(Servo_Axis_Node_4.CommonBusFault) MOV(1,EL_CTRL_4.SourceData.CommonBusFault) ,XIO(Servo_Axis_Node_4.CommonBusFault) MOV(0,EL_CTRL_4.SourceData.CommonBusFault) ,XIC(Servo_Axis_Node_4.PreChargeOverloadFault) MOV(1,EL_CTRL_4.SourceData.PreChargeOverloadFault) ,XIO(Servo_Axis_Node_4.PreChargeOverloadFault) MOV(0,EL_CTRL_4.SourceData.PreChargeOverloadFault) ,XIC(Servo_Axis_Node_4.GroundShortFault) MOV(1,EL_CTRL_4.SourceData.GroundShortFault) ,XIO(Servo_Axis_Node_4.GroundShortFault) MOV(0,EL_CTRL_4.SourceData.GroundShortFault) ,XIC(Servo_Axis_Node_4.DriveHardFault) MOV(1,EL_CTRL_4.SourceData.DriveHardFault) ,XIO(Servo_Axis_Node_4.DriveHardFault) MOV(0,EL_CTRL_4.SourceData.DriveHardFault) ,XIC(Servo_Axis_Node_4.OverSpeedFault) MOV(1,EL_CTRL_4.SourceData.OverSpeedFault) ,XIO(Servo_Axis_Node_4.OverSpeedFault) MOV(0,EL_CTRL_4.SourceData.OverSpeedFault) ,XIC(Servo_Axis_Node_4.OverloadFault) MOV(1,EL_CTRL_4.SourceData.OverloadFault) ,XIO(Servo_Axis_Node_4.OverloadFault) MOV(0,EL_CTRL_4.SourceData.OverloadFault) ,XIC(Servo_Axis_Node_4.DriveOvertempFault) MOV(1,EL_CTRL_4.SourceData.DriveOvertempFault) ,XIO(Servo_Axis_Node_4.DriveOvertempFault) MOV(0,EL_CTRL_4.SourceData.DriveOvertempFault) ,XIC(Servo_Axis_Node_4.MotorOvertempFault) MOV(1,EL_CTRL_4.SourceData.MotorOvertempFault) ,XIO(Servo_Axis_Node_4.MotorOvertempFault) MOV(0,EL_CTRL_4.SourceData.MotorOvertempFault) ,XIC(Servo_Axis_Node_4.DriveCoolingFault) MOV(1,EL_CTRL_4.SourceData.DriveCoolingFault) ,XIO(Servo_Axis_Node_4.DriveCoolingFault) MOV(0,EL_CTRL_4.SourceData.DriveCoolingFault) ,XIC(Servo_Axis_Node_4.DriveControlVoltageFault) MOV(1,EL_CTRL_4.SourceData.DriveControlVoltageFault) ,XIO(Servo_Axis_Node_4.DriveControlVoltageFault) MOV(0,EL_CTRL_4.SourceData.DriveControlVoltageFault) ,XIC(Servo_Axis_Node_4.FeedbackFault) MOV(1,EL_CTRL_4.SourceData.FeedbackFault) ,XIO(Servo_Axis_Node_4.FeedbackFault) MOV(0,EL_CTRL_4.SourceData.FeedbackFault) ,XIC(Servo_Axis_Node_4.CommutationFault) MOV(1,EL_CTRL_4.SourceData.CommutationFault) ,XIO(Servo_Axis_Node_4.CommutationFault) MOV(0,EL_CTRL_4.SourceData.CommutationFault) ,XIC(Servo_Axis_Node_4.DriveOvercurrentFault) MOV(1,EL_CTRL_4.SourceData.DriveOvercurrentFault) ,XIO(Servo_Axis_Node_4.DriveOvercurrentFault) MOV(0,EL_CTRL_4.SourceData.DriveOvercurrentFault) ,XIC(Servo_Axis_Node_4.DriveOvervoltageFault) MOV(1,EL_CTRL_4.SourceData.DriveOvervoltageFault) ,XIO(Servo_Axis_Node_4.DriveOvervoltageFault) MOV(0,EL_CTRL_4.SourceData.DriveOvervoltageFault) ,XIC(Servo_Axis_Node_4.DriveUndervoltageFault) MOV(1,EL_CTRL_4.SourceData.DriveUndervoltageFault) ,XIO(Servo_Axis_Node_4.DriveUndervoltageFault) MOV(0,EL_CTRL_4.SourceData.DriveUndervoltageFault) ,XIC(Servo_Axis_Node_4.PowerPhaseLossFault) MOV(1,EL_CTRL_4.SourceData.PowerPhaseLossFault) ,XIO(Servo_Axis_Node_4.PowerPhaseLossFault) MOV(0,EL_CTRL_4.SourceData.PowerPhaseLossFault) ,XIC(Servo_Axis_Node_4.PositionErrorFault) MOV(1,EL_CTRL_4.SourceData.PositionErrorFault) ,XIO(Servo_Axis_Node_4.PositionErrorFault) MOV(0,EL_CTRL_4.SourceData.PositionErrorFault) ,XIC(Servo_Axis_Node_4.SERCOSFault) MOV(1,EL_CTRL_4.SourceData.SERCOSFault) ,XIO(Servo_Axis_Node_4.SERCOSFault) MOV(0,EL_CTRL_4.SourceData.SERCOSFault) ,MOV(70,EL_CTRL_4.Index) ];
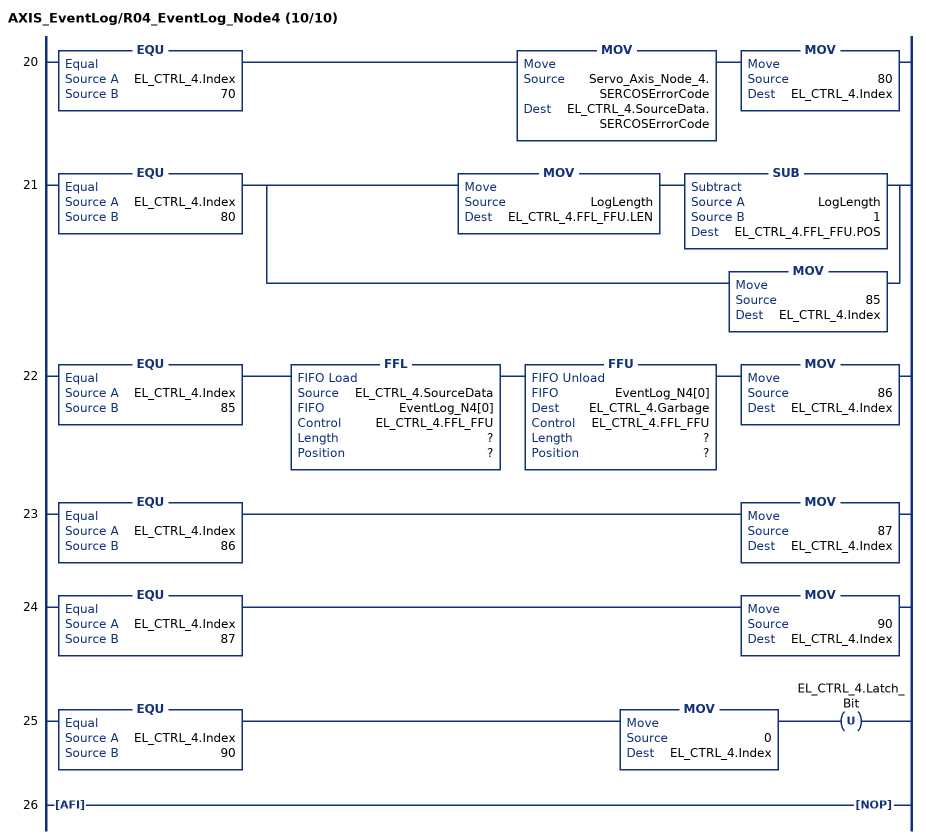
   20: EQU(EL_CTRL_4.Index,70)MOV(Servo_Axis_Node_4.SERCOSErrorCode,EL_CTRL_4.SourceData.SERCOSErrorCode)MOV(80,EL_CTRL_4.Index);
   21: EQU(EL_CTRL_4.Index,80)[MOV(LogLength,EL_CTRL_4.FFL_FFU.LEN) SUB(LogLength,1,EL_CTRL_4.FFL_FFU.POS) ,MOV(85,EL_CTRL_4.Index) ];
   22: EQU(EL_CTRL_4.Index,85)FFL(EL_CTRL_4.SourceData,EventLog_N4[0],EL_CTRL_4.FFL_FFU,?,?)FFU(EventLog_N4[0],EL_CTRL_4.Garbage,EL_CTRL_4.FFL_FFU,?,?)MOV(86,EL_CTRL_4.Index);
   23: EQU(EL_CTRL_4.Index,86)MOV(87,EL_CTRL_4.Index);
   24: EQU(EL_CTRL_4.Index,87)MOV(90,EL_CTRL_4.Index);
   25: EQU(EL_CTRL_4.Index,90)MOV(0,EL_CTRL_4.Index)OTU(EL_CTRL_4.Latch_Bit);
   26: AFI()NOP();
END_ROUTINE
